// TIA Portal project "babu_hmiBasics" (V15)

(* hardware
DEVICE "HMI_1"  KTP400 Basic PN
   slot 0: "HMI_1"  KTP400 Basic PN  6AV2 123-2DB03-0AX0  15.0.0.0
   slot 1: "HMI_RT_1"  KTP400 Basic PN  6AV2 123-2DB03-0AX0  15.0.0.0
   slot 5: "HMI_1.IE_CP_1"  PROFINET Interface  15.0.0.0
      slot 1: "PROFINET Interface_1"  PROFINET Interface
         slot 1: "Port_1"  Port
DEVICE "S7-1200 station_1"  S7-1200 Station
   slot 0: "Rack_0"  S7-1200 Rack  Rack  V1.0
   slot 1: "PLC_1"  CPU 1214C DC/DC/DC  6ES7 214-1AG40-0XB0  V4.2
*)

// ===== PLC "PLC_1"  CPU 1214C DC/DC/DC =====

VAR_GLOBAL   // PLC tag table "Default tag table"
   "START PB" AT %M0.0 : Bool;
   "START PB MEM" AT %M0.1 : Bool;
   "MEMORY" AT %M0.2 : Bool;
   "STOP PB" AT %M0.3 : Bool;
   "MOTOR" AT %Q0.0 : Bool;
END_VAR

ORGANIZATION_BLOCK "Main"   // OB1, LAD, ProgramCycle
TITLE = "Main Program Sweep (Cycle)"
{ S7_Optimized_Access := 'TRUE' }
VERSION : 0.1
   VAR_INPUT
      Initial_Call : Bool;   // Initial call of this OB
      Remanence : Bool;   // =True, if remanent data are available
   END_VAR
BEGIN

REGION Network 1
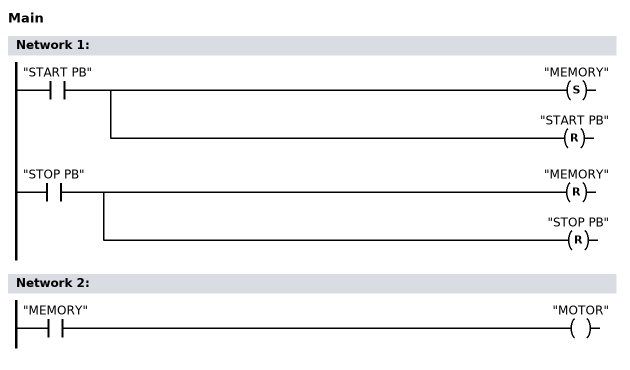
   RUNG wire#powerrail
      Contact( "START PB" )
      wire#w1
      S_Coil( "MEMORY" )
   END_RUNG
   RUNG wire#w1
      R_Coil( "START PB" )
   END_RUNG
   RUNG wire#powerrail
      Contact( "STOP PB" )
      wire#w2
      R_Coil( "MEMORY" )
   END_RUNG
   RUNG wire#w2
      R_Coil( "STOP PB" )
   END_RUNG
   // the same network as SCL:
   IF "START PB" THEN
       "MEMORY" := TRUE;
       "START PB" := FALSE;
   END_IF;
   IF "STOP PB" THEN
       "MEMORY" := FALSE;
       "STOP PB" := FALSE;
   END_IF;
END_REGION

REGION Network 2
   RUNG wire#powerrail
      Contact( "MEMORY" )
      Coil( "MOTOR" )
   END_RUNG
   // the same network as SCL:
   "MOTOR" := "MEMORY";
END_REGION
END_ORGANIZATION_BLOCK

(* ===== HMI "HMI_RT_1" =====
system functions are stored by id; their names below are inferred from use
connection "HMI_Connection_1": ETHERNET, SMART_S7_1200_OMS

HMI tags "Default tag table"
   "Tag_ScreenNumber" : UInt, internal
   "MEMORY" : Bool = PLC MEMORY AT %M0.2, 1 s
   "START PB" : Bool = PLC "START PB" AT %M0.0, 1 s
   "STOP PB" : Bool = PLC "STOP PB" AT %M0.3, 1 s

Template "Template_1" 480x272
   Button "Exit" at 388,227 size 63x44; TextOff 'Exit'; PictureOff "ExitRuntime_KTP400_Basic_PN_TR"; PictureOn "ExitRuntime_KTP400_Basic_PN_TR"
      on Release: StopRuntime(0)
   Button "Template_Button" at 268,227 size 63x44; TextOff 'Text'
   Button "Alarms" at 148,227 size 63x44; TextOff 'Alarms'; PictureOff "AlarmDisplay_KTP400_Basic_PN_TR"; PictureOn "AlarmDisplay_KTP400_Basic_PN_TR"
      on Release: function_ef3f5d25("Alarm window_Unacknowledged", -1)
   Button "Start screen" at 28,227 size 63x44; TextOff 'Start screen'; PictureOff "NavigateHome_KTP400_Basic_PN_TR"; PictureOn "NavigateHome_KTP400_Basic_PN_TR"
      on Release: ActivateScreen("Root screen", 0)
   SymbolicIOField "Symbolic_IO_Field_Screen" at 82,8 size 311x29; TextOff '0'; TextOn '1'; TextList "TextList_ScreenNames"
      ProcessValue <- "Tag_ScreenNumber"
      on Change: ActivateScreenByNumber("Tag_ScreenNumber", 0)
   DateTimeField "HmiScreenItemData" at 395,22 size 85x22
   DateTimeField "HmiScreenItemData_1" at 395,0 size 85x22
   GraphicView "Logo" at 0,0 size 80x45; Picture "Logo of HMI_1"

screen "Root screen" 480x272, template "Template_1"
   on GenerateScreen: SetTag("Tag_ScreenNumber", 1)
   Button "Button_1" at 26,75 size 176x32; TextOff 'START PUSH BUTTON'
      on Press: SetBit("START PB")
      on Release: ResetBit("START PB")
      Appearance <- "START PB"
   Button "Button_2" at 26,144 size 176x32; TextOff 'STOP PUSH BUTTON'
      on Press: SetBit("STOP PB")
      on Release: ResetBit("STOP PB")
      Appearance <- "STOP PB"
   Circle "Circle_1" at 327,79 size 97x97
      Appearance <- "MEMORY"
   TextField "Text field_1" at 347,116 size 57x22; Text 'MOTOR'
*)